// TwinCAT 3 PLC project TrimSaw
// ProgramVersion: 3.1.4023.0
// libraries:
//   Tc2_Standard, * (Beckhoff Automation GmbH)
//   Tc2_System, * (Beckhoff Automation GmbH)
//   Tc3_Module, * (Beckhoff Automation GmbH)
// project tree:
//   DUTs/ ST_Set.TcDUT
//   GVLs/ Deck1.TcGVL, Deck2.TcGVL, Deck3.TcGVL, Deck4.TcGVL, HMI.TcGVL, Inputs.TcGVL, Outputs.TcGVL
//   / PlcTask.TcTTO
//   POUs/ HMI_Controls.TcPOU, MAIN.TcPOU
//   POUs/Trim_Saw/ Trim_Saw_Pre.TcPOU, Trim_Saw_Step.TcPOU
// real-time tasks:
//   TASK PlcTask: cycle T#10ms, priority 20, ADS port 350
// I/O:
//   DEVICE Device 1 (EtherCAT), AmsNetId 10.22.66.127.2.1
//     Term 1 (EK1200) [EK1200-5000 EtherCAT Power supply (2A E-Bus)]
//       Term 2 (EL6070) [EL6070 1Ch. Licensing-Terminal]
//       Term 3 (EL3142) [EL3142 2Ch. Ana Input 0-20mA]
//       Term 4 (EL9011) [EL9011 End Terminal]
//   DEVICE Device 6 (EtherCAT), AmsNetId 10.22.66.127.7.1
//     Term 5 (EK1100-0008) [EK1100-0008 EtherCAT Coupler M8 (2A E-Bus)]
//       Term 6 (EL2634) [EL2634 4Ch. Relay Output, NO (250V AC / 30V DC)]
//       Term 7 (EL2634) [EL2634 4Ch. Relay Output, NO (250V AC / 30V DC)]
//       Term 8 (EL2634) [EL2634 4Ch. Relay Output, NO (250V AC / 30V DC)]
//       Term 9 (EL2634) [EL2634 4Ch. Relay Output, NO (250V AC / 30V DC)]
//       Term 10 (EL2634) [EL2634 4Ch. Relay Output, NO (250V AC / 30V DC)]
//       Term 9 (EL9011) [EL9011 End Terminal]
//     Box 18 (ATV320 EtherCAT) [ATV320 EtherCAT V1.13]
//     Box 19 (ATV320 EtherCAT) [ATV320 EtherCAT V1.13]
// variable links:
//   TrimSaw/TrimSaw Instance <-> Device 1 (EtherCAT)/Term 1 (EK1200)/Term 3 (EL3142)
//     PlcTask Inputs/Inputs.i_iBoardThickness[0] <-> AI Standard Channel 1/Value
//     PlcTask Inputs/Inputs.i_iBoardThickness[1] <-> AI Standard Channel 2/Value
//   TrimSaw/TrimSaw Instance <-> Device 6 (EtherCAT)/Term 5 (EK1100-0008)/Term 6 (EL2634)
//     PlcTask Outputs/Outputs.q_xDeck5DropSawFour <-> Channel 3/Output
//     PlcTask Outputs/Outputs.q_xDeck5DropSawSix <-> Channel 4/Output
//     PlcTask Outputs/Outputs.q_xDeck5DropSawTwo <-> Channel 2/Output
//     PlcTask Outputs/Outputs.q_xDeck5DropSawZero <-> Channel 1/Output
//   TrimSaw/TrimSaw Instance <-> Device 6 (EtherCAT)/Term 5 (EK1100-0008)/Term 7 (EL2634)
//     PlcTask Outputs/Outputs.q_xDeck5DropSawEight <-> Channel 1/Output
//     PlcTask Outputs/Outputs.q_xDeck5DropSawFourteen <-> Channel 4/Output
//     PlcTask Outputs/Outputs.q_xDeck5DropSawTen <-> Channel 2/Output
//     PlcTask Outputs/Outputs.q_xDeck5DropSawTwelve <-> Channel 3/Output
//   TrimSaw/TrimSaw Instance <-> Device 6 (EtherCAT)/Term 5 (EK1100-0008)/Term 8 (EL2634)
//     PlcTask Outputs/Outputs.q_xDeck5DropSawEighteen <-> Channel 2/Output
//     PlcTask Outputs/Outputs.q_xDeck5DropSawSixteen <-> Channel 1/Output

CONFIGURATION TrimSaw
    RESOURCE PLC ON TwinCAT3
        TASK PlcTask(INTERVAL := T#10ms, PRIORITY := 20);
        PROGRAM MAIN WITH PlcTask : MAIN;
    END_RESOURCE
END_CONFIGURATION

// ---- DUTs/ST_Set.TcDUT
TYPE ST_Set :
STRUCT
stBoardSize : STRING;
stEndEven : STRING;
END_STRUCT
END_TYPE

// ---- GVLs/Deck1.TcGVL
VAR_GLOBAL
	//Deck 1
	//Drive inputs
	ATV_State_D1							AT	%I*		: WORD; //Drive state
	ATV_TPDO_Input1_Status_Word_D1			AT	%I*		: WORD;	//Status Word From Drive
	iVelocityRaw_D1							AT	%I*		: INT;	//Velocity From Drive - Address 8604 - Units 1 RPM
	iTorqueRaw_D1							AT	%I*		: INT;	//Torque From Drive - Address 3205 - Units 0.1%
	uiCurrentRaw_D1							AT	%I*		: UINT;	//Current From Drive - Address 3204 - Units 0.1A
	uiVoltageRaw_D1							AT	%I*		: UINT;	//Voltage From Drive - Address 3208 - Units 1V
	uiFaultCode_D1							AT	%I*		: UINT;	//Fault Codes
	//End drive inputs	

	//Drive outputs
	ATV_RPDO_Output1_Control_Word_D1		AT	%Q*		: WORD;	//Control Word To Drive
	ATV_RPDO_Output2_Target_Velocity_D1		AT	%Q*		: WORD; //Velocity To Drive in RPM - Max Value 32767
	//End drive outputs

	//Inputs Status Word Bit Level
	xReady_To_Switch_on_D1 								: BOOL;//Bit 0
	xSwitched_ON_D1										: BOOL;//Bit 1
	xOperationEnabled_D1 								: BOOL;//Bit 2
	xFault_D1 											: BOOL;//Bit 3
	xVoltageEnabled_D1									: BOOL;//Bit 4
	xQuickStop_D1										: BOOL;//Bit 5
	xSwitchOnDisabled_D1 								: BOOL;//Bit 6
	xWarning_D1											: BOOL;//Bit 7
	xTargetReached_D1									: BOOL;//Bit 10
	xInternalLimitActive_D1								: BOOL;//Bit 11
	xDirectionofRotation_D1								: BOOL;//Bit 15	
	stFault_D1											: STRING;
	rTorqueValue_D1										: REAL;
	rCurrentValue_D1									: REAL;
	lrSpeed_D1											: LREAL;
	xEnable_D1											: BOOL; //Enable Drive Trigger
	xStart_D1											: BOOL;	//Start Trigger
	xStop_D1 											: BOOL;	//Stop Trigger
	iDirection_D1										: INT;	//Direction	Trigger
	xForward_D1											: BOOL; //Forward Trigger
	xReverse_D1											: BOOL;	//Reverse Trigger
	xReset_D1											: BOOL;	//Reset Trigger
	xInputStatus_HMI_D1									: ARRAY [0..9] OF BOOL;	//VFD Status Bits
	//End inputs Status Word Bit Level
	//End Deck 1
END_VAR

// ---- GVLs/Deck2.TcGVL
VAR_GLOBAL
	//Deck 2
	//Drive inputs
	ATV_State_D2							AT	%I*		: WORD; //Drive state
	ATV_TPDO_Input1_Status_Word_D2			AT	%I*		: WORD;	//Status Word From Drive
	iVelocityRaw_D2							AT	%I*		: INT;	//Velocity From Drive - Address 8604 - Units 1 RPM
	iTorqueRaw_D2							AT	%I*		: INT;	//Torque From Drive - Address 3205 - Units 0.1%
	uiCurrentRaw_D2							AT	%I*		: UINT;	//Current From Drive - Address 3204 - Units 0.1A
	uiVoltageRaw_D2							AT	%I*		: UINT;	//Voltage From Drive - Address 3208 - Units 1V
	uiFaultCode_D2							AT	%I*		: UINT;	//Fault Codes
	//End drive inputs	
	
	//Drive outputs
	ATV_RPDO_Output1_Control_Word_D2		AT	%Q*		: WORD;	//Control Word To Drive
	ATV_RPDO_Output2_Target_Velocity_D2		AT	%Q*		: WORD; //Velocity To Drive in RPM - Max Value 32767
	//End drive outputs

	//Inputs Status Word Bit Level
	xReady_To_Switch_on_D2 								: BOOL;//Bit 0
	xSwitched_ON_D2										: BOOL;//Bit 1
	xOperationEnabled_D2 								: BOOL;//Bit 2
	xFault_D2 											: BOOL;//Bit 3
	xVoltageEnabled_D2									: BOOL;//Bit 4
	xQuickStop_D2										: BOOL;//Bit 5
	xSwitchOnDisabled_D2 								: BOOL;//Bit 6
	xWarning_D2											: BOOL;//Bit 7
	xTargetReached_D2									: BOOL;//Bit 10
	xInternalLimitActive_D2								: BOOL;//Bit 11
	xDirectionofRotation_D2								: BOOL;//Bit 15	
	stFault_D2											: STRING;
	rTorqueValue_D2										: REAL;
	rCurrentValue_D2									: REAL;
	lrSpeed_D2											: LREAL;
	xEnable_D2											: BOOL; //Enable Drive Trigger
	xStart_D2											: BOOL;	//Start Trigger
	xStop_D2 											: BOOL;	//Stop Trigger
	iDirection_D2										: INT;	//Direction	Trigger
	xForward_D2											: BOOL; //Forward Trigger
	xReverse_D2											: BOOL;	//Reverse Trigger
	xReset_D2											: BOOL;	//Reset Trigger
	xInputStatus_HMI_D2									: ARRAY [0..9] OF BOOL;	//VFD Status Bits
	//End inputs Status Word Bit Level
	//End Deck 1
END_VAR

// ---- GVLs/Deck3.TcGVL
VAR_GLOBAL
	//Deck 1
	//Drive inputs
	ATV_State_D3							AT	%I*		: WORD; //Drive state
	ATV_TPDO_Input1_Status_Word_D3			AT	%I*		: WORD;	//Status Word From Drive
	iVelocityRaw_D3							AT	%I*		: INT;	//Velocity From Drive - Address 8604 - Units 1 RPM
	iTorqueRaw_D3							AT	%I*		: INT;	//Torque From Drive - Address 3205 - Units 0.1%
	uiCurrentRaw_D3							AT	%I*		: UINT;	//Current From Drive - Address 3204 - Units 0.1A
	uiVoltageRaw_D3							AT	%I*		: UINT;	//Voltage From Drive - Address 3208 - Units 1V
	uiFaultCode_D3							AT	%I*		: UINT;	//Fault Codes
	//End drive inputs	
	
	//Drive outputs
	ATV_RPDO_Output1_Control_Word_D3		AT	%Q*		: WORD;	//Control Word To Drive
	ATV_RPDO_Output2_Target_Velocity_D3		AT	%Q*		: WORD; //Velocity To Drive in RPM - Max Value 32767
	//End drive outputs

	//Inputs Status Word Bit Level
	xReady_To_Switch_on_D3 								: BOOL;//Bit 0
	xSwitched_ON_D3										: BOOL;//Bit 1
	xOperationEnabled_D3 								: BOOL;//Bit 2
	xFault_D3 											: BOOL;//Bit 3
	xVoltageEnabled_D3									: BOOL;//Bit 4
	xQuickStop_D3										: BOOL;//Bit 5
	xSwitchOnDisabled_D3 								: BOOL;//Bit 6
	xWarning_D3											: BOOL;//Bit 7
	xTargetReached_D3									: BOOL;//Bit 10
	xInternalLimitActive_D3								: BOOL;//Bit 11
	xDirectionofRotation_D3								: BOOL;//Bit 15	
	stFault_D3											: STRING;
	rTorqueValue_D3										: REAL;
	rCurrentValue_D3									: REAL;
	lrSpeed_D3											: LREAL;
	xEnable_D3											: BOOL; //Enable Drive Trigger
	xStart_D3											: BOOL;	//Start Trigger
	xStop_D3 											: BOOL;	//Stop Trigger
	iDirection_D3										: INT;	//Direction	Trigger
	xForward_D3											: BOOL; //Forward Trigger
	xReverse_D3											: BOOL;	//Reverse Trigger
	xReset_D3											: BOOL;	//Reset Trigger
	xInputStatus_HMI_D3									: ARRAY [0..9] OF BOOL;	//VFD Status Bits
	//End inputs Status Word Bit Level
	//End Deck 1
END_VAR

// ---- GVLs/Deck4.TcGVL
VAR_GLOBAL
	//Deck 1
	//Drive inputs
	ATV_State_D4							AT	%I*		: WORD; //Drive state
	ATV_TPDO_Input1_Status_Word_D4			AT	%I*		: WORD;	//Status Word From Drive
	iVelocityRaw_D4							AT	%I*		: INT;	//Velocity From Drive - Address 8604 - Units 1 RPM
	iTorqueRaw_D4							AT	%I*		: INT;	//Torque From Drive - Address 3205 - Units 0.1%
	uiCurrentRaw_D4							AT	%I*		: UINT;	//Current From Drive - Address 3204 - Units 0.1A
	uiVoltageRaw_D4							AT	%I*		: UINT;	//Voltage From Drive - Address 3208 - Units 1V
	uiFaultCode_D4							AT	%I*		: UINT;	//Fault Codes
	//End drive inputs	
	
	//Drive outputs
	ATV_RPDO_Output1_Control_Word_D4		AT	%Q*		: WORD;	//Control Word To Drive
	ATV_RPDO_Output2_Target_Velocity_D4		AT	%Q*		: WORD; //Velocity To Drive in RPM - Max Value 32767
	//End drive outputs

	//Inputs Status Word Bit Level
	xReady_To_Switch_on_D4 								: BOOL;//Bit 0
	xSwitched_ON_D4										: BOOL;//Bit 1
	xOperationEnabled_D4 								: BOOL;//Bit 2
	xFault_D4 											: BOOL;//Bit 3
	xVoltageEnabled_D4									: BOOL;//Bit 4
	xQuickStop_D4										: BOOL;//Bit 5
	xSwitchOnDisabled_D4 								: BOOL;//Bit 6
	xWarning_D4											: BOOL;//Bit 7
	xTargetReached_D4									: BOOL;//Bit 10
	xInternalLimitActive_D4								: BOOL;//Bit 11
	xDirectionofRotation_D4								: BOOL;//Bit 15	
	stFault_D4											: STRING;
	rTorqueValue_D4										: REAL;
	rCurrentValue_D4									: REAL;
	lrSpeed_D4											: LREAL;
	xEnable_D4											: BOOL; //Enable Drive Trigger
	xStart_D4											: BOOL;	//Start Trigger
	xStop_D4 											: BOOL;	//Stop Trigger
	iDirection_D4										: INT;	//Direction	Trigger
	xForward_D4											: BOOL; //Forward Trigger
	xReverse_D4											: BOOL;	//Reverse Trigger
	xReset_D4											: BOOL;	//Reset Trigger
	xInputStatus_HMI_D4									: ARRAY [0..9] OF BOOL;	//VFD Status Bits
	//End inputs Status Word Bit Level
	//End Deck 1
END_VAR

// ---- GVLs/HMI.TcGVL
{attribute 'qualified_only'}
VAR_GLOBAL
lrVFD_Set_Velocity 			: ARRAY [0..3] OF LREAL;
lrVFD_Actual_Velocity 		: ARRAY [0..3] OF LREAL;

xButton_Board_Size 			: ARRAY [0..9] OF BOOL;
xButton_Board_Size_HMI 		: ARRAY [0..9] OF BOOL;
stButton_Board_Size 		: ARRAY [0..9] OF STRING;

xButton_Even_End 			: ARRAY [0..2] OF BOOL;
xButton_Even_End_HMI 		: ARRAY [0..2] OF BOOL;
stButton_Even_End_HMI 		: ARRAY [0..2] OF STRING;

NextSets 					: ARRAY[0..9] OF ST_Set;
lrCurrentThickenss 			: ARRAY[0..1] OF LREAL;
rPieceCount 				: REAL;
xClearSets 					: BOOL;

stVFDIndicator				: ARRAY[0..9] OF STRING;

stStatusMessage_HMI			: STRING;

xStartStopButton			: BOOL;
stStartStopButton			: STRING;

xSlowFastButton				: BOOL;
stSlowFastButton			: STRING;

xResetButton				: BOOL;


//Recipe parameters
rSlowSpeed					: ARRAY [0..3] OF REAL;
rFastSpeed					: ARRAY [0..3] OF REAL;
lrLaserScaling				: ARRAY[0..1] OF LREAL;
lrLaserOffset				: ARRAY[0..1] OF LREAL;
lrBoardThicknessLimit		: LREAL;
//End Recipe Parameters

//VFD Jog buttons 
xJogForward_HMI					: ARRAY [0..3] OF BOOL;
xJogReverse_HMI					: ARRAY [0..3] OF BOOL;

//Outputs 
stOutputs_Text					: ARRAY [0..17] OF STRING;
xOutputs						: ARRAY [0..17] OF BOOL;

END_VAR

// ---- GVLs/Inputs.TcGVL
{attribute 'qualified_only'}
VAR_GLOBAL
	i_xSawEntryPhotoEye					AT %I*	: BOOL;
	i_xSawExitPhotoEye					AT %I*	: BOOL;
	
	i_iBoardThickness					AT %I*	: ARRAY[0..1] OF INT;	
	
	i_xFootSwitch						AT %I*	: BOOL;
	
	//DEMO
	i_xJoyStickButton1					AT %I*	: BOOL;
	i_xJoyStickButton2					AT %I*	: BOOL;
	//END DEMO
END_VAR

// ---- GVLs/Outputs.TcGVL
{attribute 'qualified_only'}
VAR_GLOBAL
	q_xDeck3Stopper					AT %Q*	: BOOL;
	q_xDeck4PressureRoller			AT %Q*	: BOOL;
	q_xDeck4ZeroEndZero				AT %Q*	: BOOL;
	q_xDeck4ZeroEndMinusOne			AT %Q*	: BOOL;
	q_xDeck4ZeroEndMinusTwo			AT %Q*	: BOOL;
	q_xDeck4ZeroEndMotor			AT %Q*	: BOOL;
	q_xDeck5DropSawZero				AT %Q*	: BOOL;
	q_xDeck5DropSawTwo				AT %Q*	: BOOL;
	q_xDeck5DropSawFour				AT %Q*	: BOOL;
	q_xDeck5DropSawSix				AT %Q*	: BOOL;
	q_xDeck5DropSawEight			AT %Q*	: BOOL;
	q_xDeck5DropSawTen				AT %Q*	: BOOL;
	q_xDeck5DropSawTwelve			AT %Q*	: BOOL;
	q_xDeck5DropSawFourteen			AT %Q*	: BOOL;
	q_xDeck5DropSawSixteen			AT %Q*	: BOOL;
	q_xDeck5DropSawEighteen			AT %Q*	: BOOL;
	q_xDeck6Tipple					AT %Q*	: BOOL;
END_VAR

// ---- POUs/MAIN.TcPOU
PROGRAM MAIN
VAR
	arr_FaultCodes					: ARRAY [0..110] OF STRING; 
	lrSpeed_HMI_D1					: LREAL;
	
	stRecipeName					: STRING;
	
	
	//Remove after demo
	fb_DRAND						: Drand;
	fb_DRAND2						: Drand;
	fb_DRAND3						: Drand;
	fb_DRAND4						: Drand;
END_VAR

HMI_Controls();
Trim_Saw_Pre();
Trim_Saw_Step();
Deck_1();
Deck_2();
Deck_3();
Deck_4();
FaultCodes();

stRecipeName := 'TrimSaw';

ACTION Deck_1:
//Inputs from VFD
(*xInputStatus_HMI_D1[0] := xReady_To_Switch_on_D1 := BIT_TO_BOOL (ATV_TPDO_Input1_Status_Word_D1.0); 
xInputStatus_HMI_D1[1] := xSwitched_ON_D1:= BIT_TO_BOOL (ATV_TPDO_Input1_Status_Word_D1.1); 
xInputStatus_HMI_D1[2] := xOperationEnabled_D1 := BIT_TO_BOOL (ATV_TPDO_Input1_Status_Word_D1.2); 
xInputStatus_HMI_D1[3] := xFault_D1 := BIT_TO_BOOL (ATV_TPDO_Input1_Status_Word_D1.3); 
xInputStatus_HMI_D1[4] := xVoltageEnabled_D1 := BIT_TO_BOOL (ATV_TPDO_Input1_Status_Word_D1.4); 
xInputStatus_HMI_D1[5] := xQuickStop_D1:= BIT_TO_BOOL (ATV_TPDO_Input1_Status_Word_D1.5); 
xInputStatus_HMI_D1[6] := xSwitchOnDisabled_D1 := BIT_TO_BOOL (ATV_TPDO_Input1_Status_Word_D1.6); 
xInputStatus_HMI_D1[7] := xWarning_D1:= BIT_TO_BOOL (ATV_TPDO_Input1_Status_Word_D1.7); 
xInputStatus_HMI_D1[8] := xTargetReached_D1:= BIT_TO_BOOL (ATV_TPDO_Input1_Status_Word_D1.10); 
xInputStatus_HMI_D1[9] := xInternalLimitActive_D1:= BIT_TO_BOOL (ATV_TPDO_Input1_Status_Word_D1.11); *)
xDirectionofRotation_D1:= BIT_TO_BOOL (ATV_TPDO_Input1_Status_Word_D1.15);
rTorqueValue_D1 := iTorqueRaw_D1/10.0;
rCurrentValue_D1 := uiCurrentRaw_D1/10.0;
stFault_D1 := arr_FaultCodes[uiFaultCode_D1];

//Actual Speed
//HMI.lrVFD_Actual_Velocity[0] := iVelocityRaw_D1;	**********Remove comment after demo	

//************************************************************Remove After Demo
fb_DRAND(Seed:= 10, Num=>HMI.lrVFD_Actual_Velocity[0]);
HMI.lrVFD_Actual_Velocity[0] := HMI.lrVFD_Actual_Velocity[0] + 100;
IF HMI.lrVFD_Actual_Velocity[0] > 101 THEN
	HMI.lrVFD_Actual_Velocity[0] := 0;
END_IF
//************************************************************End Remove After Demo

//Speed
ATV_RPDO_Output2_Target_Velocity_D1 := LREAL_TO_WORD (lrSpeed_D1);

//Direction
IF xForward_D1 THEN
	iDirection_D1 := 0;	
	xReverse_D1 := FALSE;
ELSIF xReverse_D1 THEN
	iDirection_D1 := 1;
	xForward_D1 := FALSE;
END_IF

//Enable Control Word
IF xEnable_D1 AND NOT xStart_D1 THEN
	ATV_RPDO_Output1_Control_Word_D1.0 := 0;//Switch ON
	ATV_RPDO_Output1_Control_Word_D1.1 := 1;//Enable Voltage
	ATV_RPDO_Output1_Control_Word_D1.2 := 1;//Quick Stop
	ATV_RPDO_Output1_Control_Word_D1.3 := 0;//Enable Operation
	ATV_RPDO_Output1_Control_Word_D1.11 := INT_TO_BIT (iDirection_D1);//Direction
END_IF

//Start Control Word
IF xEnable_D1 AND xStart_D1 THEN
	ATV_RPDO_Output1_Control_Word_D1.0 := 1;//Switch ON
	ATV_RPDO_Output1_Control_Word_D1.1 := 1;//Enable Voltage
	ATV_RPDO_Output1_Control_Word_D1.2 := 1;//Quick Stop
	ATV_RPDO_Output1_Control_Word_D1.3 := 1;//Enable Operation
END_IF

//Stop Control Word
IF xEnable_D1 AND xStop_D1 THEN
	xStart_D1 := FALSE;
	ATV_RPDO_Output1_Control_Word_D1.0 := 0;//Switch ON
	ATV_RPDO_Output1_Control_Word_D1.1 := 1;//Enable Voltage
	ATV_RPDO_Output1_Control_Word_D1.2 := 1;//Quick Stop
	ATV_RPDO_Output1_Control_Word_D1.3 := 0;//Enable Operation
END_IF

//Reset Control Word
IF xReset_D1 THEN
	ATV_RPDO_Output1_Control_Word_D1.7 := 1;//Reset Fault
ELSE 
	ATV_RPDO_Output1_Control_Word_D1.7 := 0;//Reset Fault
END_IF

//Reset if not enabled
IF NOT xEnable_D1 THEN
	ATV_RPDO_Output1_Control_Word_D1.0 := 0;//Switch ON
	ATV_RPDO_Output1_Control_Word_D1.1 := 0;//Enable Voltage
	ATV_RPDO_Output1_Control_Word_D1.2 := 0;//Quick Stop
	ATV_RPDO_Output1_Control_Word_D1.3 := 0;//Enable Operation
	xStart_D1 := FALSE;
	xStop_D1 := FALSE;
END_IF
END_ACTION

ACTION Deck_2:
//Inputs from VFD
(*xInputStatus_HMI_D2[0] := xReady_To_Switch_on_D2 := BIT_TO_BOOL (ATV_TPDO_Input1_Status_Word_D2.0); 
xInputStatus_HMI_D2[1] := xSwitched_ON_D2:= BIT_TO_BOOL (ATV_TPDO_Input1_Status_Word_D2.1); 
xInputStatus_HMI_D2[2] := xOperationEnabled_D2 := BIT_TO_BOOL (ATV_TPDO_Input1_Status_Word_D2.2); 
xInputStatus_HMI_D2[3] := xFault_D2 := BIT_TO_BOOL (ATV_TPDO_Input1_Status_Word_D2.3); 
xInputStatus_HMI_D2[4] := xVoltageEnabled_D2 := BIT_TO_BOOL (ATV_TPDO_Input1_Status_Word_D2.4); 
xInputStatus_HMI_D2[5] := xQuickStop_D2:= BIT_TO_BOOL (ATV_TPDO_Input1_Status_Word_D2.5); 
xInputStatus_HMI_D2[6] := xSwitchOnDisabled_D2 := BIT_TO_BOOL (ATV_TPDO_Input1_Status_Word_D2.6); 
xInputStatus_HMI_D2[7] := xWarning_D2:= BIT_TO_BOOL (ATV_TPDO_Input1_Status_Word_D2.7); 
xInputStatus_HMI_D2[8] := xTargetReached_D2:= BIT_TO_BOOL (ATV_TPDO_Input1_Status_Word_D2.10); 
xInputStatus_HMI_D2[9] := xInternalLimitActive_D2:= BIT_TO_BOOL (ATV_TPDO_Input1_Status_Word_D2.11); *)
xDirectionofRotation_D2:= BIT_TO_BOOL (ATV_TPDO_Input1_Status_Word_D2.15);
rTorqueValue_D2 := iTorqueRaw_D2/10.0;
rCurrentValue_D2 := uiCurrentRaw_D2/10.0;
stFault_D2 := arr_FaultCodes[uiFaultCode_D2];

//Actual Speed
//HMI.lrVFD_Actual_Velocity[1] := iVelocityRaw_D2;	**********Remove comment after demo

//************************************************************Remove After Demo
fb_DRAND2(Seed:= 4, Num=>HMI.lrVFD_Actual_Velocity[1]);
HMI.lrVFD_Actual_Velocity[1] := HMI.lrVFD_Actual_Velocity[1] + 100;
IF HMI.lrVFD_Actual_Velocity[1] > 101 THEN
	HMI.lrVFD_Actual_Velocity[1] := 0;
END_IF
//************************************************************End Remove After Demo

//Speed
ATV_RPDO_Output2_Target_Velocity_D2 := LREAL_TO_WORD (lrSpeed_D2);

//Direction
IF xForward_D2 THEN
	iDirection_D2 := 0;	
	xReverse_D2 := FALSE;
ELSIF xReverse_D2 THEN
	iDirection_D2 := 1;
	xForward_D2 := FALSE;
END_IF

//Enable Control Word
IF xEnable_D2 AND NOT xStart_D2 THEN
	ATV_RPDO_Output1_Control_Word_D2.0 := 0;//Switch ON
	ATV_RPDO_Output1_Control_Word_D2.1 := 1;//Enable Voltage
	ATV_RPDO_Output1_Control_Word_D2.2 := 1;//Quick Stop
	ATV_RPDO_Output1_Control_Word_D2.3 := 0;//Enable Operation
	ATV_RPDO_Output1_Control_Word_D2.11 := INT_TO_BIT (iDirection_D2);//Direction
END_IF

//Start Control Word
IF xEnable_D2 AND xStart_D2 THEN
	ATV_RPDO_Output1_Control_Word_D2.0 := 1;//Switch ON
	ATV_RPDO_Output1_Control_Word_D2.1 := 1;//Enable Voltage
	ATV_RPDO_Output1_Control_Word_D2.2 := 1;//Quick Stop
	ATV_RPDO_Output1_Control_Word_D2.3 := 1;//Enable Operation
END_IF

//Stop Control Word
IF xEnable_D2 AND xStop_D2 THEN
	xStart_D2 := FALSE;
	ATV_RPDO_Output1_Control_Word_D2.0 := 0;//Switch ON
	ATV_RPDO_Output1_Control_Word_D2.1 := 1;//Enable Voltage
	ATV_RPDO_Output1_Control_Word_D2.2 := 1;//Quick Stop
	ATV_RPDO_Output1_Control_Word_D2.3 := 0;//Enable Operation
END_IF

//Reset Control Word
IF xReset_D2 THEN
	ATV_RPDO_Output1_Control_Word_D2.7 := 1;//Reset Fault
ELSE 
	ATV_RPDO_Output1_Control_Word_D2.7 := 0;//Reset Fault
END_IF

//Reset if not enabled
IF NOT xEnable_D2 THEN
	ATV_RPDO_Output1_Control_Word_D2.0 := 0;//Switch ON
	ATV_RPDO_Output1_Control_Word_D2.1 := 0;//Enable Voltage
	ATV_RPDO_Output1_Control_Word_D2.2 := 0;//Quick Stop
	ATV_RPDO_Output1_Control_Word_D2.3 := 0;//Enable Operation
	xStart_D2 := FALSE;
	xStop_D2 := FALSE;
END_IF
END_ACTION

ACTION Deck_3:
//Inputs from VFD
(*xInputStatus_HMI_D3[0] := xReady_To_Switch_on_D3 := BIT_TO_BOOL (ATV_TPDO_Input1_Status_Word_D3.0); 
xInputStatus_HMI_D3[1] := xSwitched_ON_D3:= BIT_TO_BOOL (ATV_TPDO_Input1_Status_Word_D3.1); 
xInputStatus_HMI_D3[2] := xOperationEnabled_D3 := BIT_TO_BOOL (ATV_TPDO_Input1_Status_Word_D3.2); 
xInputStatus_HMI_D3[3] := xFault_D3 := BIT_TO_BOOL (ATV_TPDO_Input1_Status_Word_D3.3); 
xInputStatus_HMI_D3[4] := xVoltageEnabled_D3 := BIT_TO_BOOL (ATV_TPDO_Input1_Status_Word_D3.4); 
xInputStatus_HMI_D3[5] := xQuickStop_D3:= BIT_TO_BOOL (ATV_TPDO_Input1_Status_Word_D3.5); 
xInputStatus_HMI_D3[6] := xSwitchOnDisabled_D3 := BIT_TO_BOOL (ATV_TPDO_Input1_Status_Word_D3.6); 
xInputStatus_HMI_D3[7] := xWarning_D3:= BIT_TO_BOOL (ATV_TPDO_Input1_Status_Word_D3.7); 
xInputStatus_HMI_D3[8] := xTargetReached_D3:= BIT_TO_BOOL (ATV_TPDO_Input1_Status_Word_D3.10); 
xInputStatus_HMI_D3[9] := xInternalLimitActive_D3:= BIT_TO_BOOL (ATV_TPDO_Input1_Status_Word_D3.11); *)
xDirectionofRotation_D3:= BIT_TO_BOOL (ATV_TPDO_Input1_Status_Word_D3.15);
rTorqueValue_D3 := iTorqueRaw_D3/10.0;
rCurrentValue_D3 := uiCurrentRaw_D3/10.0;
stFault_D3 := arr_FaultCodes[uiFaultCode_D3];

//Actual Speed
//HMI.lrVFD_Actual_Velocity[2] := iVelocityRaw_D3;	**********Remove comment after demo	

//************************************************************Remove After Demo
fb_DRAND3(Seed:= 3, Num=>HMI.lrVFD_Actual_Velocity[2]);
HMI.lrVFD_Actual_Velocity[2] := HMI.lrVFD_Actual_Velocity[2] + 100;
IF HMI.lrVFD_Actual_Velocity[2] > 101 THEN
	HMI.lrVFD_Actual_Velocity[2] := 0;
END_IF
//************************************************************End Remove After Demo

//Speed
ATV_RPDO_Output2_Target_Velocity_D3 := LREAL_TO_WORD (lrSpeed_D3);

//Direction
IF xForward_D3 THEN
	iDirection_D3 := 0;	
	xReverse_D3 := FALSE;
ELSIF xReverse_D3 THEN
	iDirection_D3 := 1;
	xForward_D3 := FALSE;
END_IF

//Enable Control Word
IF xEnable_D3 AND NOT xStart_D3 THEN
	ATV_RPDO_Output1_Control_Word_D3.0 := 0;//Switch ON
	ATV_RPDO_Output1_Control_Word_D3.1 := 1;//Enable Voltage
	ATV_RPDO_Output1_Control_Word_D3.2 := 1;//Quick Stop
	ATV_RPDO_Output1_Control_Word_D3.3 := 0;//Enable Operation
	ATV_RPDO_Output1_Control_Word_D3.11 := INT_TO_BIT (iDirection_D3);//Direction
END_IF

//Start Control Word
IF xEnable_D3 AND xStart_D3 THEN
	ATV_RPDO_Output1_Control_Word_D3.0 := 1;//Switch ON
	ATV_RPDO_Output1_Control_Word_D3.1 := 1;//Enable Voltage
	ATV_RPDO_Output1_Control_Word_D3.2 := 1;//Quick Stop
	ATV_RPDO_Output1_Control_Word_D3.3 := 1;//Enable Operation
END_IF

//Stop Control Word
IF xEnable_D3 AND xStop_D3 THEN
	xStart_D3 := FALSE;
	ATV_RPDO_Output1_Control_Word_D3.0 := 0;//Switch ON
	ATV_RPDO_Output1_Control_Word_D3.1 := 1;//Enable Voltage
	ATV_RPDO_Output1_Control_Word_D3.2 := 1;//Quick Stop
	ATV_RPDO_Output1_Control_Word_D3.3 := 0;//Enable Operation
END_IF

//Reset Control Word
IF xReset_D3 THEN
	ATV_RPDO_Output1_Control_Word_D3.7 := 1;//Reset Fault
ELSE 
	ATV_RPDO_Output1_Control_Word_D3.7 := 0;//Reset Fault
END_IF

//Reset if not enabled
IF NOT xEnable_D3 THEN
	ATV_RPDO_Output1_Control_Word_D3.0 := 0;//Switch ON
	ATV_RPDO_Output1_Control_Word_D3.1 := 0;//Enable Voltage
	ATV_RPDO_Output1_Control_Word_D3.2 := 0;//Quick Stop
	ATV_RPDO_Output1_Control_Word_D3.3 := 0;//Enable Operation
	xStart_D3 := FALSE;
	xStop_D3 := FALSE;
END_IF
END_ACTION

ACTION Deck_4:
//Inputs from VFD
(*xInputStatus_HMI_D4[0] := xReady_To_Switch_on_D4 := BIT_TO_BOOL (ATV_TPDO_Input1_Status_Word_D4.0); 
xInputStatus_HMI_D4[1] := xSwitched_ON_D4:= BIT_TO_BOOL (ATV_TPDO_Input1_Status_Word_D4.1); 
xInputStatus_HMI_D4[2] := xOperationEnabled_D4 := BIT_TO_BOOL (ATV_TPDO_Input1_Status_Word_D4.2); 
xInputStatus_HMI_D4[3] := xFault_D4 := BIT_TO_BOOL (ATV_TPDO_Input1_Status_Word_D4.3); 
xInputStatus_HMI_D4[4] := xVoltageEnabled_D4 := BIT_TO_BOOL (ATV_TPDO_Input1_Status_Word_D4.4); 
xInputStatus_HMI_D4[5] := xQuickStop_D4:= BIT_TO_BOOL (ATV_TPDO_Input1_Status_Word_D4.5); 
xInputStatus_HMI_D4[6] := xSwitchOnDisabled_D4 := BIT_TO_BOOL (ATV_TPDO_Input1_Status_Word_D4.6); 
xInputStatus_HMI_D4[7] := xWarning_D4:= BIT_TO_BOOL (ATV_TPDO_Input1_Status_Word_D4.7); 
xInputStatus_HMI_D4[8] := xTargetReached_D4:= BIT_TO_BOOL (ATV_TPDO_Input1_Status_Word_D4.10); 
xInputStatus_HMI_D4[9] := xInternalLimitActive_D4:= BIT_TO_BOOL (ATV_TPDO_Input1_Status_Word_D4.11); *)
xDirectionofRotation_D4:= BIT_TO_BOOL (ATV_TPDO_Input1_Status_Word_D4.15);
rTorqueValue_D4 := iTorqueRaw_D4/10.0;
rCurrentValue_D4 := uiCurrentRaw_D4/10.0;
stFault_D4 := arr_FaultCodes[uiFaultCode_D4];

//Actual Speed
//HMI.lrVFD_Actual_Velocity[3] := iVelocityRaw_D4;	**********Remove comment after demo

//************************************************************Remove After Demo
fb_DRAND4(Seed:= 2, Num=>HMI.lrVFD_Actual_Velocity[3]);
HMI.lrVFD_Actual_Velocity[3] := HMI.lrVFD_Actual_Velocity[3] + 100;
IF HMI.lrVFD_Actual_Velocity[3] > 101 THEN
	HMI.lrVFD_Actual_Velocity[3] := 0;
END_IF
//************************************************************End Remove After Demo

//Speed
ATV_RPDO_Output2_Target_Velocity_D4 := LREAL_TO_WORD (lrSpeed_D4);

//Direction
IF xForward_D4 THEN
	iDirection_D4 := 0;	
	xReverse_D4 := FALSE;
ELSIF xReverse_D4 THEN
	iDirection_D4 := 1;
	xForward_D4 := FALSE;
END_IF

//Enable Control Word
IF xEnable_D4 AND NOT xStart_D4 THEN
	ATV_RPDO_Output1_Control_Word_D4.0 := 0;//Switch ON
	ATV_RPDO_Output1_Control_Word_D4.1 := 1;//Enable Voltage
	ATV_RPDO_Output1_Control_Word_D4.2 := 1;//Quick Stop
	ATV_RPDO_Output1_Control_Word_D4.3 := 0;//Enable Operation
	ATV_RPDO_Output1_Control_Word_D4.11 := INT_TO_BIT (iDirection_D4);//Direction
END_IF

//Start Control Word
IF xEnable_D4 AND xStart_D4 THEN
	ATV_RPDO_Output1_Control_Word_D4.0 := 1;//Switch ON
	ATV_RPDO_Output1_Control_Word_D4.1 := 1;//Enable Voltage
	ATV_RPDO_Output1_Control_Word_D4.2 := 1;//Quick Stop
	ATV_RPDO_Output1_Control_Word_D4.3 := 1;//Enable Operation
END_IF

//Stop Control Word
IF xEnable_D4 AND xStop_D4 THEN
	xStart_D4 := FALSE;
	ATV_RPDO_Output1_Control_Word_D4.0 := 0;//Switch ON
	ATV_RPDO_Output1_Control_Word_D4.1 := 1;//Enable Voltage
	ATV_RPDO_Output1_Control_Word_D4.2 := 1;//Quick Stop
	ATV_RPDO_Output1_Control_Word_D4.3 := 0;//Enable Operation
END_IF

//Reset Control Word
IF xReset_D4 THEN
	ATV_RPDO_Output1_Control_Word_D4.7 := 1;//Reset Fault
ELSE 
	ATV_RPDO_Output1_Control_Word_D4.7 := 0;//Reset Fault
END_IF

//Reset if not enabled
IF NOT xEnable_D4 THEN
	ATV_RPDO_Output1_Control_Word_D4.0 := 0;//Switch ON
	ATV_RPDO_Output1_Control_Word_D4.1 := 0;//Enable Voltage
	ATV_RPDO_Output1_Control_Word_D4.2 := 0;//Quick Stop
	ATV_RPDO_Output1_Control_Word_D4.3 := 0;//Enable Operation
	xStart_D4 := FALSE;
	xStop_D4 := FALSE;
END_IF
END_ACTION

ACTION FaultCodes:
arr_FaultCodes[0]:='No faults';
arr_FaultCodes[2]:='EEprom control fault';
arr_FaultCodes[3]:='Incorrect configuration';
arr_FaultCodes[4]:='Invalid config parameters';
arr_FaultCodes[5]:='Modbus coms fault';
arr_FaultCodes[6]:='Com Internal link fault';
arr_FaultCodes[7]:='Network fault';
arr_FaultCodes[8]:='External fault logic input';
arr_FaultCodes[9]:='Overcurrent fault';
arr_FaultCodes[10]:='Precharge';
arr_FaultCodes[11]:='Speed feedback loss';
arr_FaultCodes[12]:='Output speed <> ref';
arr_FaultCodes[16]:='Drive overheating fault';
arr_FaultCodes[17]:='Motor overload fault';
arr_FaultCodes[18]:='DC bus overvoltage fault';
arr_FaultCodes[19]:='Supply overvoltage fault';
arr_FaultCodes[20]:='1 motor phase loss fault';
arr_FaultCodes[21]:='Supply phase loss fault';
arr_FaultCodes[22]:='Supply undervolt fault';
arr_FaultCodes[23]:='Motor short circuit';
arr_FaultCodes[24]:='Motor overspeed fault';
arr_FaultCodes[25]:='Auto-tuning fault';
arr_FaultCodes[26]:='Rating error';
arr_FaultCodes[27]:='Incompatible control card';
arr_FaultCodes[28]:='Internal coms link fault';
arr_FaultCodes[29]:='Internal manu zone fault';
arr_FaultCodes[30]:='EEprom power fault';
arr_FaultCodes[32]:='Ground short circuit';
arr_FaultCodes[33]:='3 motor phase loss fault';
arr_FaultCodes[34]:='Comms fault CANopen';
arr_FaultCodes[35]:='Brake control fault';
arr_FaultCodes[38]:='External fault comms';
arr_FaultCodes[41]:='Brake feedback fault';
arr_FaultCodes[42]:='PC coms fault';
arr_FaultCodes[44]:='Torque/current limit fault';
arr_FaultCodes[45]:='HMI coms fault';
arr_FaultCodes[49]:='LI6=PTC failed';
arr_FaultCodes[50]:='LI6=PTC overheat fault';
arr_FaultCodes[51]:='Internal I measure fault';
arr_FaultCodes[52]:='Internal i/p volt circuit flt';
arr_FaultCodes[53]:='Internal temperature fault';
arr_FaultCodes[54]:='IGBT overheat fault';
arr_FaultCodes[55]:='IGBT short circuit fault';
arr_FaultCodes[56]:='Motor short circuit';
arr_FaultCodes[58]:='Output cont close fault';
arr_FaultCodes[59]:='Output cont open fault';
arr_FaultCodes[64]:='input contactor';
arr_FaultCodes[67]:='IGBT desaturation';
arr_FaultCodes[68]:='Internal option fault';
arr_FaultCodes[69]:='Internal- CPU ';
arr_FaultCodes[71]:='AI3 4-20mA loss';
arr_FaultCodes[73]:='Cards pairing';
arr_FaultCodes[76]:='Dynamic load fault';
arr_FaultCodes[77]:='Interrupted config.';
arr_FaultCodes[99]:='Channel switching fault';
arr_FaultCodes[100]:='Process Underlaod Fault';
arr_FaultCodes[101]:='Process Overload Fault';
arr_FaultCodes[105]:='Angle error';
arr_FaultCodes[107]:='Safety fault';
arr_FaultCodes[108]:='FB fault';
arr_FaultCodes[109]:='FB stop fault';
END_ACTION

END_PROGRAM

// ---- POUs/HMI_Controls.TcPOU
PROGRAM HMI_Controls
VAR
	
	xTriggerOneShot : ARRAY [0..9] OF BOOL;
	xTriggerOneShot_1 : ARRAY [0..2] OF BOOL;
	xTriggerOneShot_2 : ARRAY [0..2] OF BOOL;
	xTriggerOneShot_3				: BOOL;
	x: INT;
	y: INT;	
	z: INT;
	i: INT;
	h: INT;
	j: INT;
	b: INT;
	c: INT;
	r_trigger_1: R_Trig;
	//Remove after demo
	tDemoTimer: TON;
	tDemoTimer2: Ton;
	tDemoTimer3: TON;
	t : int;
	
	

	xIOPage: BOOL;
END_VAR

FOR Y := 0 TO 9 DO
	IF HMI.NextSets[y].stBoardSize = '' THEN
		EXIT;
	END_IF
END_FOR

//Board Size Selection
FOR x := 0 TO 9 DO
	IF HMI.xButton_Board_Size_HMI[x] AND NOT xTriggerOneShot[x]THEN
		IF NOT HMI.xButton_Board_Size_HMI[4] THEN
			b := 0;
		END_IF
		IF NOT HMI.xButton_Board_Size[x] THEN
			//HMI.xButton_Board_Size[x] := TRUE;
			xTriggerOneShot[x]:= TRUE;
			HMI.NextSets[y].stBoardSize := HMI.stButton_Board_Size[x];
			FOR j := 0 TO 2 DO
				IF HMI.xButton_Even_End[j] THEN
					HMI.NextSets[y].stEndEven := HMI.stButton_Even_End_HMI[j];
				END_IF
			END_FOR
			HMI.xButton_Even_End[0] := TRUE;
			y :=y + 1;
		ELSIF HMI.xButton_Board_Size[x] THEN
			HMI.xButton_Board_Size[x] := FALSE;	
			xTriggerOneShot[x]:= TRUE;
		END_IF
	ELSIF NOT HMI.xButton_Board_Size_HMI[x] AND xTriggerOneShot[x]THEN
		xTriggerOneShot[x]:= FALSE;
	END_IF
END_FOR

r_trigger_1 (CLK:= HMI.xButton_Board_Size_HMI[4]);
IF r_trigger_1.q THEN
	b := b + 1;
	IF b >=  3 THEN
		FOR c := 0 TO 9 DO
			HMI.NextSets[c].stEndEven := '0';
		END_FOR
	END_IF		
END_IF
// End Board Size Selection

//Even End Selection
FOR i := 0 TO 2 DO
	IF HMI.xButton_Even_End_HMI[i] AND NOT xTriggerOneShot_1[i]THEN
		IF NOT HMI.xButton_Even_End[i] THEN
			HMI.xButton_Even_End[i] := TRUE;
			xTriggerOneShot_1[i] := TRUE;	
		ELSIF HMI.xButton_Even_End[i] THEN						
			HMI.xButton_Even_End[i] := FALSE;	
			xTriggerOneShot_1[i] := TRUE;					
		END_IF
	ELSIF NOT HMI.xButton_Even_End_HMI[i] AND xTriggerOneShot_1[i]THEN	
		xTriggerOneShot_1[i] := FALSE;
	END_IF
END_FOR


HMI.stButton_Even_End_HMI[0] := '0';
HMI.stButton_Even_End_HMI[1] := '-1';
HMI.stButton_Even_End_HMI[2] := '-2';

HMI.stButton_Board_Size[0] := '8';
HMI.stButton_Board_Size[1] := '10';
HMI.stButton_Board_Size[2] := '12';
HMI.stButton_Board_Size[3] := '14'; 
HMI.stButton_Board_Size[4] := '16';
HMI.stButton_Board_Size[5] := '18';
HMI.stButton_Board_Size[6] := 'Trash';
HMI.stButton_Board_Size[7] := 'Saws Up';

			


IF NOT HMI.xButton_Even_End[0] AND NOT HMI.xButton_Even_End[1] AND NOT HMI.xButton_Even_End[2] THEN
	HMI.xButton_Even_End[0]:= TRUE;
END_IF
IF HMI.xButton_Even_End[0] AND NOT xTriggerOneShot_2[0] THEN
	HMI.xButton_Even_End[1] :=
	HMI.xButton_Even_End[2] := FALSE;
	xTriggerOneShot_2[0] := TRUE;
	xTriggerOneShot_2[1] := 
	xTriggerOneShot_2[2] := FALSE;
ELSIF HMI.xButton_Even_End[1] AND NOT xTriggerOneShot_2[1]THEN
	HMI.xButton_Even_End[0] :=
	HMI.xButton_Even_End[2] := FALSE;
	xTriggerOneShot_2[1] := TRUE;
	xTriggerOneShot_2[0] := 
	xTriggerOneShot_2[2] := FALSE;
ELSIF HMI.xButton_Even_End[2] AND NOT xTriggerOneShot_2[2]THEN
	HMI.xButton_Even_End[0] :=
	HMI.xButton_Even_End[1] := FALSE;
	xTriggerOneShot_2[2] := TRUE;
	xTriggerOneShot_2[0] := 
	xTriggerOneShot_2[1] := FALSE;
END_IF		 

		
IF HMI.xClearSets THEN
	FOR z := 0 TO 9 DO
		HMI.NextSets[z].stEndEven := '';
		HMI.NextSets[z].stBoardSize:= '';
		HMI.xButton_Board_Size[z] := FALSE;	
		b := 0;
	END_FOR
	FOR h := 0 TO 2 DO
		HMI.xButton_Even_End[h] := FALSE;	
	END_FOR
	y := 0;
END_IF

HMI.stVFDIndicator[0] :='Ready To Switch ON';
HMI.stVFDIndicator[1] :='Switched ON';
HMI.stVFDIndicator[2] :='Operation Enabled';
HMI.stVFDIndicator[3] :='Fault';
HMI.stVFDIndicator[4] :='Voltage Enabled';
HMI.stVFDIndicator[5] :='Quick Stop';
HMI.stVFDIndicator[6] :='Switch ON Disabled';
HMI.stVFDIndicator[7] :='Warning';
HMI.stVFDIndicator[8] :='Target Reached';
HMI.stVFDIndicator[9] :='INTERNAL LIMIT Active';

//Control buttons logic
IF HMI.xStartStopButton THEN
	HMI.stStartStopButton := 'Stop';
ELSE
	HMI.stStartStopButton := 'Start';
END_IF

IF HMI.xSlowFastButton THEN
	HMI.stSlowFastButton := 'Fast';
ELSE
	HMI.stSlowFastButton := 'Slow';
END_IF
//End control buttons logic




//Outputs

(*IF xIOPage THEN
	HMI.xOutputs[0]:=Outputs.q_xDeck3Stopper;
	HMI.xOutputs[1]:=Outputs.q_xDeck4PressureRoller;
	HMI.xOutputs[2]:=Outputs.q_xDeck4ZeroEndZero;
	HMI.xOutputs[3]:=Outputs.q_xDeck4ZeroEndMinusOne;
	HMI.xOutputs[4]:=Outputs.q_xDeck4ZeroEndMinusTwo;
	HMI.xOutputs[5]:=Outputs.q_xDeck4ZeroEndMotor;
	HMI.xOutputs[6]:=Outputs.q_xDeck5DropSawZero;
	HMI.xOutputs[7]:=Outputs.q_xDeck5DropSawTwo;
	HMI.xOutputs[8]:=Outputs.q_xDeck5DropSawFour;
	HMI.xOutputs[9]:=Outputs.q_xDeck5DropSawSix;
	HMI.xOutputs[10]:=Outputs.q_xDeck5DropSawEight;
	HMI.xOutputs[11]:=Outputs.q_xDeck5DropSawTen;
	HMI.xOutputs[12]:=Outputs.q_xDeck5DropSawTwelve;
	HMI.xOutputs[13]:=Outputs.q_xDeck5DropSawFourteen;
	HMI.xOutputs[14]:=Outputs.q_xDeck5DropSawSixteen;
	HMI.xOutputs[15]:=Outputs.q_xDeck5DropSawEighteen;
	HMI.xOutputs[16]:=Outputs.q_xDeck6Tipple;
END_IF*)



HMI.xOutputs[0]:=Outputs.q_xDeck3Stopper;
HMI.xOutputs[1]:=Outputs.q_xDeck4PressureRoller;
HMI.xOutputs[2]:=Outputs.q_xDeck4ZeroEndZero;
HMI.xOutputs[3]:=Outputs.q_xDeck4ZeroEndMinusOne;
HMI.xOutputs[4]:=Outputs.q_xDeck4ZeroEndMinusTwo;
HMI.xOutputs[5]:=Outputs.q_xDeck4ZeroEndMotor;
HMI.xOutputs[6]:=Outputs.q_xDeck5DropSawZero;
HMI.xOutputs[7]:=Outputs.q_xDeck5DropSawTwo;
HMI.xOutputs[8]:=Outputs.q_xDeck5DropSawFour;
HMI.xOutputs[9]:=Outputs.q_xDeck5DropSawSix;
HMI.xOutputs[10]:=Outputs.q_xDeck5DropSawEight;
HMI.xOutputs[11]:=Outputs.q_xDeck5DropSawTen;
HMI.xOutputs[12]:=Outputs.q_xDeck5DropSawTwelve;
HMI.xOutputs[13]:=Outputs.q_xDeck5DropSawFourteen;
HMI.xOutputs[14]:=Outputs.q_xDeck5DropSawSixteen;
HMI.xOutputs[15]:=Outputs.q_xDeck5DropSawEighteen;
HMI.xOutputs[16]:=Outputs.q_xDeck6Tipple;


HMI.stOutputs_Text[0]:='Deck 3 Stopper';
HMI.stOutputs_Text[1]:='Deck 4 Pressure Roller';
HMI.stOutputs_Text[2]:='Deck 4 Zero End Zero';
HMI.stOutputs_Text[3]:='Deck 4 Zero End Minus One';
HMI.stOutputs_Text[4]:='Deck 4 Zero End Minus Two';
HMI.stOutputs_Text[5]:='Deck 4 Zero End Motor';
HMI.stOutputs_Text[6]:='Deck 5 Drop Saw Zero';
HMI.stOutputs_Text[7]:='Deck 5 Drop Saw Two';
HMI.stOutputs_Text[8]:='Deck 5 Drop Saw Four';
HMI.stOutputs_Text[9]:='Deck 5 Drop Saw Six';
HMI.stOutputs_Text[10]:='Deck 5 Drop Saw Eight';
HMI.stOutputs_Text[11]:='Deck 5 Drop Saw Ten';
HMI.stOutputs_Text[12]:='Deck 5 Drop Saw Twelve';
HMI.stOutputs_Text[13]:='Deck 5 Drop Saw Fourteen';
HMI.stOutputs_Text[14]:='Deck 5 Drop Saw Sixteen';
HMI.stOutputs_Text[15]:='Deck 5 Drop Saw Eighteen';
HMI.stOutputs_Text[16]:='Deck 6 Tipple';

//*******************************Remove After Demo
(*tDemoTimer(PT := T#2S);
tDemoTimer3(PT := T#2S);
IF Trim_Saw_Step.iStep = (0 OR 50) AND HMI.NextSets[0].stBoardSize <> ''THEN
	tDemoTimer.IN := TRUE;
END_IF

IF tDemoTimer.Q THEN	
	IF HMI.rPieceCount < 300 THEN
		HMI.rPieceCount := HMI.rPieceCount + 1;
	ELSE
		HMI.rPieceCount := 0;
	END_IF
	IF HMI.lrCurrentThickenss[0] < 6.1 THEN
		//HMI.lrCurrentThickenss := HMI.lrCurrentThickenss + 1.2;
	ELSE
		//HMI.lrCurrentThickenss := 1;
	END_IF
	tDemoTimer.IN := FALSE;
	Inputs.i_xSawEntryPhotoEye := TRUE;
	tDemoTimer3.IN := TRUE;
END_IF

IF tDemoTimer3.Q THEN
	tDemoTimer3.IN := FALSE;
	Inputs.i_xSawExitPhotoEye := TRUE;
END_IF

tDemoTimer2(PT := T#2S);
tDemoTimer2.IN := TRUE;
IF tDemoTimer2.Q THEN
	IF t < 10 THEN
		xInputStatus_HMI_D1[t]:= TRUE;
		xInputStatus_HMI_D2[t]:= TRUE;
		xInputStatus_HMI_D3[t]:= TRUE;
		xInputStatus_HMI_D4[t]:= TRUE;
		IF t > 0 THEN
			xInputStatus_HMI_D1[t-1]:= FALSE;
			xInputStatus_HMI_D2[t-1]:= FALSE;
			xInputStatus_HMI_D3[t-1]:= FALSE;
			xInputStatus_HMI_D4[t-1]:= FALSE;
		END_IF	
		t := t + 1;
	ELSE
		xInputStatus_HMI_D1[9]:= FALSE;
		xInputStatus_HMI_D2[9]:= FALSE;
		xInputStatus_HMI_D3[9]:= FALSE;
		xInputStatus_HMI_D4[9]:= FALSE;
		t := 0;
	END_IF
	tDemoTimer2.IN := FALSE;
END_IF*)


IF Inputs.i_xJoyStickButton1 THEN
	Inputs.i_xSawEntryPhotoEye := TRUE;
ELSE
	Inputs.i_xSawEntryPhotoEye := FALSE;
END_IF

IF Inputs.i_xJoyStickButton2 THEN
	Inputs.i_xSawExitPhotoEye := TRUE;
ELSE
	Inputs.i_xSawExitPhotoEye := FALSE;
END_IF











//*******************************End Remove After Demo

END_PROGRAM

// ---- POUs/Trim_Saw/Trim_Saw_Pre.TcPOU
PROGRAM Trim_Saw_Pre
VAR
	tonSawEntryPhotoEye				: TON;
	tonSawExitPhotoEye				: TON;
	tonFootSwitch					: TON;
	lrBoardThickness				: ARRAY[0..1] OF LREAL;
END_VAR

tonSawEntryPhotoEye(IN := Inputs.i_xSawEntryPhotoEye, PT := T#50MS);
tonSawExitPhotoEye(IN := Inputs.i_xSawExitPhotoEye, PT := T#50MS);
tonFootSwitch(IN := Inputs.i_xFootSwitch, PT := T#50MS);

IF HMI.lrLaserScaling[0] <> 0 THEN
	lrBoardThickness[0] := Inputs.i_iBoardThickness[0] / HMI.lrLaserScaling[0] + HMI.lrLaserOffset[0];
	HMI.lrCurrentThickenss[0] := lrBoardThickness[0];
END_IF

IF HMI.lrLaserScaling[1] <> 0 THEN
	lrBoardThickness[1] := Inputs.i_iBoardThickness[1] / HMI.lrLaserScaling[1] + HMI.lrLaserOffset[1];
	HMI.lrCurrentThickenss[1] := lrBoardThickness[1];
END_IF

IF tonFootSwitch.Q THEN
	Outputs.q_xDeck3Stopper := TRUE;
ELSE
	Outputs.q_xDeck3Stopper := FALSE;
END_IF

IF HMI.xSlowFastButton THEN
	//Set conveyor speed to slow
ELSE
	//Set conveyor speed to fast
END_IF

//For Demo
//lrBoardThickness := HMI.lrCurrentThickenss;

IF tonSawEntryPhotoEye.Q THEN
	Inputs.i_xSawEntryPhotoEye := FALSE;
END_IF

IF tonSawExitPhotoEye.Q THEN
	Inputs.i_xSawExitPhotoEye := FALSE;
END_IF

END_PROGRAM

// ---- POUs/Trim_Saw/Trim_Saw_Step.TcPOU
PROGRAM Trim_Saw_Step
VAR
	iStep						: INT;
	iCount						: INT;
	xError						: BOOL;
END_VAR

IF HMI.xStartStopButton THEN
	CASE iStep OF
		0: //Stack loaded
			HMI.stStatusMessage_HMI := 'Waiting for first board in stack to be loaded.';
			IF HMI.NextSets[0].stBoardSize <> '' THEN
				iStep := 10;
			END_IF
		10: //Set Even Ender Stop
			HMI.stStatusMessage_HMI := 'Setting even ender position.';
			IF HMI.NextSets[0].stEndEven = '0' THEN
				Outputs.q_xDeck4ZeroEndZero := TRUE;
				Outputs.q_xDeck4ZeroEndMinusOne := FALSE;
				Outputs.q_xDeck4ZeroEndMinusTwo := FALSE;
			ELSIF HMI.NextSets[0].stEndEven = '-1' THEN
				Outputs.q_xDeck4ZeroEndZero := FALSE;
				Outputs.q_xDeck4ZeroEndMinusOne := TRUE;
				Outputs.q_xDeck4ZeroEndMinusTwo := FALSE;
			ELSIF HMI.NextSets[0].stEndEven = '-2' THEN
				Outputs.q_xDeck4ZeroEndZero := FALSE;
				Outputs.q_xDeck4ZeroEndMinusOne := FALSE;
				Outputs.q_xDeck4ZeroEndMinusTwo := TRUE;
			ELSE
				//Error
				HMI.stStatusMessage_HMI := 'Error: Even ender position not possible.';
				iStep := 99;
				RETURN;
			END_IF
			iStep := 20;
		20: //Lower even ender pressure roller and turn on even ender motor
			HMI.stStatusMessage_HMI := 'Lowering even ender pressure roller and turning on even ender motor.';
			Outputs.q_xDeck4PressureRoller := TRUE;
			Outputs.q_xDeck4ZeroEndMotor := TRUE;
			iStep := 30;
		30: //Thickness okay
			HMI.stStatusMessage_HMI := 'Checking board thickness.';
			IF Trim_Saw_Pre.lrBoardThickness[0] >= HMI.lrBoardThicknessLimit THEN
				HMI.NextSets[0].stBoardSize := 'Saws Up';
				//Set tipple
				//Clear stack for this board?				
			END_IF
			iStep := 40;
		40: //Lower appropriate saws
			HMI.stStatusMessage_HMI := 'Lowering appropriate saws.';
			IF HMI.NextSets[0].stBoardSize <> 'Trash' THEN
				Outputs.q_xDeck5DropSawZero := TRUE;
				Outputs.q_xDeck5DropSawTwo := FALSE;
				Outputs.q_xDeck5DropSawFour := TRUE;
				Outputs.q_xDeck5DropSawSix := FALSE;
				Outputs.q_xDeck5DropSawEight := TRUE;
				Outputs.q_xDeck5DropSawTen := FALSE;
				Outputs.q_xDeck5DropSawTwelve := TRUE;
				Outputs.q_xDeck5DropSawFourteen := FALSE;
				Outputs.q_xDeck5DropSawSixteen := TRUE;
				Outputs.q_xDeck5DropSawEighteen := FALSE;
			ELSIF HMI.NextSets[0].stBoardSize <> 'Saws Up' THEN
				Outputs.q_xDeck5DropSawZero := FALSE;
				Outputs.q_xDeck5DropSawTwo := FALSE;
				Outputs.q_xDeck5DropSawFour := FALSE;
				Outputs.q_xDeck5DropSawSix := FALSE;
				Outputs.q_xDeck5DropSawEight := FALSE;
				Outputs.q_xDeck5DropSawTen := FALSE;
				Outputs.q_xDeck5DropSawTwelve := FALSE;
				Outputs.q_xDeck5DropSawFourteen := FALSE;
				Outputs.q_xDeck5DropSawSixteen := FALSE;
				Outputs.q_xDeck5DropSawEighteen := FALSE;
			ELSIF HMI.NextSets[0].stBoardSize <> '2' THEN
				Outputs.q_xDeck5DropSawZero := TRUE;
				Outputs.q_xDeck5DropSawTwo := TRUE;
				Outputs.q_xDeck5DropSawFour := FALSE;
				Outputs.q_xDeck5DropSawSix := FALSE;
				Outputs.q_xDeck5DropSawEight := FALSE;
				Outputs.q_xDeck5DropSawTen := FALSE;
				Outputs.q_xDeck5DropSawTwelve := FALSE;
				Outputs.q_xDeck5DropSawFourteen := FALSE;
				Outputs.q_xDeck5DropSawSixteen := FALSE;
				Outputs.q_xDeck5DropSawEighteen := FALSE;
			ELSIF HMI.NextSets[0].stBoardSize <> '4' THEN
				Outputs.q_xDeck5DropSawZero := TRUE;
				Outputs.q_xDeck5DropSawTwo := FALSE;
				Outputs.q_xDeck5DropSawFour := TRUE;
				Outputs.q_xDeck5DropSawSix := FALSE;
				Outputs.q_xDeck5DropSawEight := FALSE;
				Outputs.q_xDeck5DropSawTen := FALSE;
				Outputs.q_xDeck5DropSawTwelve := FALSE;
				Outputs.q_xDeck5DropSawFourteen := FALSE;
				Outputs.q_xDeck5DropSawSixteen := FALSE;
				Outputs.q_xDeck5DropSawEighteen := FALSE;
			ELSIF HMI.NextSets[0].stBoardSize <> '6' THEN
				Outputs.q_xDeck5DropSawZero := TRUE;
				Outputs.q_xDeck5DropSawTwo := FALSE;
				Outputs.q_xDeck5DropSawFour := FALSE;
				Outputs.q_xDeck5DropSawSix := TRUE;
				Outputs.q_xDeck5DropSawEight := FALSE;
				Outputs.q_xDeck5DropSawTen := FALSE;
				Outputs.q_xDeck5DropSawTwelve := FALSE;
				Outputs.q_xDeck5DropSawFourteen := FALSE;
				Outputs.q_xDeck5DropSawSixteen := FALSE;
				Outputs.q_xDeck5DropSawEighteen := FALSE;
			ELSIF HMI.NextSets[0].stBoardSize <> '8' THEN
				Outputs.q_xDeck5DropSawZero := TRUE;
				Outputs.q_xDeck5DropSawTwo := FALSE;
				Outputs.q_xDeck5DropSawFour := FALSE;
				Outputs.q_xDeck5DropSawSix := FALSE;
				Outputs.q_xDeck5DropSawEight := TRUE;
				Outputs.q_xDeck5DropSawTen := FALSE;
				Outputs.q_xDeck5DropSawTwelve := FALSE;
				Outputs.q_xDeck5DropSawFourteen := FALSE;
				Outputs.q_xDeck5DropSawSixteen := FALSE;
				Outputs.q_xDeck5DropSawEighteen := FALSE;
			ELSIF HMI.NextSets[0].stBoardSize <> '10' THEN
				Outputs.q_xDeck5DropSawZero := TRUE;
				Outputs.q_xDeck5DropSawTwo := FALSE;
				Outputs.q_xDeck5DropSawFour := FALSE;
				Outputs.q_xDeck5DropSawSix := FALSE;
				Outputs.q_xDeck5DropSawEight := FALSE;
				Outputs.q_xDeck5DropSawTen := TRUE;
				Outputs.q_xDeck5DropSawTwelve := FALSE;
				Outputs.q_xDeck5DropSawFourteen := FALSE;
				Outputs.q_xDeck5DropSawSixteen := FALSE;
				Outputs.q_xDeck5DropSawEighteen := FALSE;
			ELSIF HMI.NextSets[0].stBoardSize <> '12' THEN
				Outputs.q_xDeck5DropSawZero := TRUE;
				Outputs.q_xDeck5DropSawTwo := FALSE;
				Outputs.q_xDeck5DropSawFour := FALSE;
				Outputs.q_xDeck5DropSawSix := FALSE;
				Outputs.q_xDeck5DropSawEight := FALSE;
				Outputs.q_xDeck5DropSawTen := FALSE;
				Outputs.q_xDeck5DropSawTwelve := TRUE;
				Outputs.q_xDeck5DropSawFourteen := FALSE;
				Outputs.q_xDeck5DropSawSixteen := FALSE;
				Outputs.q_xDeck5DropSawEighteen := FALSE;
			ELSIF HMI.NextSets[0].stBoardSize <> '14' THEN
				Outputs.q_xDeck5DropSawZero := TRUE;
				Outputs.q_xDeck5DropSawTwo := FALSE;
				Outputs.q_xDeck5DropSawFour := FALSE;
				Outputs.q_xDeck5DropSawSix := FALSE;
				Outputs.q_xDeck5DropSawEight := FALSE;
				Outputs.q_xDeck5DropSawTen := FALSE;
				Outputs.q_xDeck5DropSawTwelve := FALSE;
				Outputs.q_xDeck5DropSawFourteen := TRUE;
				Outputs.q_xDeck5DropSawSixteen := FALSE;
				Outputs.q_xDeck5DropSawEighteen := FALSE;
			ELSIF HMI.NextSets[0].stBoardSize <> '16' THEN
				Outputs.q_xDeck5DropSawZero := TRUE;
				Outputs.q_xDeck5DropSawTwo := FALSE;
				Outputs.q_xDeck5DropSawFour := FALSE;
				Outputs.q_xDeck5DropSawSix := FALSE;
				Outputs.q_xDeck5DropSawEight := FALSE;
				Outputs.q_xDeck5DropSawTen := FALSE;
				Outputs.q_xDeck5DropSawTwelve := FALSE;
				Outputs.q_xDeck5DropSawFourteen := FALSE;
				Outputs.q_xDeck5DropSawSixteen := TRUE;
				Outputs.q_xDeck5DropSawEighteen := FALSE;
			ELSIF HMI.NextSets[0].stBoardSize <> '18' THEN
				Outputs.q_xDeck5DropSawZero := TRUE;
				Outputs.q_xDeck5DropSawTwo := FALSE;
				Outputs.q_xDeck5DropSawFour := FALSE;
				Outputs.q_xDeck5DropSawSix := FALSE;
				Outputs.q_xDeck5DropSawEight := FALSE;
				Outputs.q_xDeck5DropSawTen := FALSE;
				Outputs.q_xDeck5DropSawTwelve := FALSE;
				Outputs.q_xDeck5DropSawFourteen := FALSE;
				Outputs.q_xDeck5DropSawSixteen := FALSE;
				Outputs.q_xDeck5DropSawEighteen := TRUE;
			ELSE
				//Error
				HMI.stStatusMessage_HMI := 'Error: Saw position not possible.';
				RETURN;
			END_IF
			iStep := 50;
		50: //Wait for entry photoeye
			HMI.stStatusMessage_HMI := 'Waiting for board to enter saw.';
			IF Trim_Saw_Pre.tonSawEntryPhotoEye.Q THEN
				iStep := 60;
			END_IF
		60: //Wait for board to exit saws
			HMI.stStatusMessage_HMI := 'Waiting for board to exit saw.';
			IF Inputs.i_xSawExitPhotoEye THEN
				FOR iCount := 0 TO 9 BY 1 DO
					IF iCount = 9 THEN
						HMI.NextSets[iCount].stBoardSize := '';
						HMI.NextSets[iCount].stEndEven := '';
					ELSE
						HMI.NextSets[iCount].stBoardSize := HMI.NextSets[iCount + 1].stBoardSize;
						HMI.NextSets[iCount].stEndEven := HMI.NextSets[iCount + 1].stEndEven;
					END_IF
				END_FOR
				iStep := 0;
			END_IF
		99: //Error
			
	END_CASE
ELSE
	Outputs.q_xDeck5DropSawZero := FALSE;
	Outputs.q_xDeck5DropSawTwo := FALSE;
	Outputs.q_xDeck5DropSawFour := FALSE;
	Outputs.q_xDeck5DropSawSix := FALSE;
	Outputs.q_xDeck5DropSawEight := FALSE;
	Outputs.q_xDeck5DropSawTen := FALSE;
	Outputs.q_xDeck5DropSawTwelve := FALSE;
	Outputs.q_xDeck5DropSawFourteen := FALSE;
	Outputs.q_xDeck5DropSawSixteen := FALSE;
	Outputs.q_xDeck5DropSawEighteen := FALSE;
	IF NOT xError THEN
		HMI.stStatusMessage_HMI := 'Waiting for start button to be pressed.';
	END_IF
END_IF

END_PROGRAM
